// TIA Portal V17 export
// export: Created 2024-08-07T21:44:10.1764301Z, ExportSetting WithDefaults, DisplayName Totally Integrated Automation Portal, DisplayVersion V17 Update 7, DisplayName TIA Portal Openness, DisplayVersion V17 Update 7, DisplayName TIA Portal Version Control Interface, DisplayVersion V17, DisplayName SINAMICS Startdrive Advanced, DisplayVersion V17 SP2, DisplayName SINAMICS Startdrive G110M, G120, G120C, G120D, G120P, G115D, DisplayVersion V17 SP2, DisplayName SINAMICS Startdrive G130, G150, S120, S150, SINAMICS MV, S210, DisplayVersion V17 SP2, DisplayName STEP 7 Professional, DisplayVersion V17 Update 7, DisplayName STEP 7 Safety, DisplayVersion V17 Update 6, DisplayName WinCC Advanced / Unified PC, DisplayVersion V17 Update 7
FUNCTION "FC_Variability" : Void   // FC2013, LAD
{ S7_Optimized_Access := 'TRUE' }
VERSION : 0.1
// V1 : Creation YM 7/04/2023
// stored: AutoNumber false, IsIECCheckEnabled false, SetENOAutomatically false, UDAEnableTagReadback false
   VAR_TEMP
      i : Int;
      j : Bool;
      result : String;
      dintLeft : DInt;
   END_VAR
BEGIN

REGION Network 1 (SCL): Convert Errors
   // FOR #i := 1 TO 32 DO
   //      "DB_Variability".ERROR[#i].%W0 := "DB_MESSAGE".ERROR_TO_HMI[(#i*2)-1];
   //      "DB_Variability".ERROR[#i].%W1 := "DB_MESSAGE".ERROR_TO_HMI[#i * 2];
   //  END_FOR;

   // FOR #i := 1 TO 32 DO
   //     // Move Error to left to remove error 0 not used on Welding cell compare standard of variability
   //     #dintLeft := SHL_DINT(IN := "DB_Variability".ERROR[#i], N := 1);
   //     //Convert Dint to String
   //     #result := "LGF_IntToString"(#dintLeft);
   //     //Convert String to wtring
   //     "DB_Variability".ERROR_TO_OPC[#i] := STRING_TO_WSTRING(#result);

   // END_FOR;
END_REGION
END_FUNCTION
